{attribute 'GeneratedUsingTerminal: EPP2816-0004-0016'}
{attribute addProperty BoxType "EPP2816-0004-0016"}
{attribute addProperty Description "EPP2816-0004 16CH. Dig. Output, Diagnostic, M16"}
{attribute addProperty Physics "YY"}
{attribute addProperty Id "DIG_Diag_Inputs_Channel_1AT %I*DIG_Diag_Inputs_Channel_584303BF8DIG_Diag_Inputs_Channel_2AT %I*DIG_Diag_Inputs_Channel_584303BF8DIG_Inputs_DeviceAT %I*DIG_Inputs_Device_E94E5BF95DIG_Output_Channel_1AT %Q*DIG_Output_Channel_28AC1A9E8DIG_Output_Channel_2AT %Q*DIG_Output_Channel_28AC1A9E8DIG_Outputs_DeviceAT %Q*DIG_Outputs_Device_36A5EF172WcStateAT %I*WcState_9091E0EB2InfoDataAT %I*InfoData_32EB74EA10"}
{attribute addProperty CRC "4193692546"}
{attribute addProperty Size "51"}
TYPE EPP2816_F9F6AB82 EXTENDS EtcSlaveBoxBase_77A0E4A7 :
STRUCT
	{attribute addProperty Name "DIG_Diag_Inputs_Channel_1"}
	DIG_Diag_Inputs_Channel_1 : DIG_Diag_Inputs_Channel_584303BF;
	{attribute addProperty Name "DIG_Diag_Inputs_Channel_2"}
	DIG_Diag_Inputs_Channel_2 : DIG_Diag_Inputs_Channel_584303BF;
	{attribute addProperty Name "DIG_Inputs_Device"}
	DIG_Inputs_Device : DIG_Inputs_Device_E94E5BF9;
	{attribute addProperty Name "DIG_Output_Channel_1"}
	DIG_Output_Channel_1 : DIG_Output_Channel_28AC1A9E;
	{attribute addProperty Name "DIG_Output_Channel_2"}
	DIG_Output_Channel_2 : DIG_Output_Channel_28AC1A9E;
	{attribute addProperty Name "DIG_Outputs_Device"}
	DIG_Outputs_Device : DIG_Outputs_Device_36A5EF17;
	{attribute addProperty Name "WcState"}
	WcState : WcState_9091E0EB;
	{attribute addProperty Name "InfoData"}
	InfoData : InfoData_32EB74EA;
END_STRUCT
END_TYPE

(* stored: Version 1.2.0.0, ProductVersion 3.1.4024.9
   DUT EPP2816_F9F6AB82: Id {d5344567-9443-45be-818b-295e5b450fe8} *)
